// TIA Portal V18 export
// export: Created 2026-06-21T12:15:02Z, ExportSetting WithDefaults
PlcWatchTable "WT_PLC1_PID_VFD"
  PlcWatchTableEntry "HMI_Sim_Mode"
  PlcWatchTableEntry "PLC1_Loi_Tong"
  PlcWatchTableEntry "PLC1_EStop_Latch"
  PlcWatchTableEntry "PLC1_Loi_Dry_Run"
  PlcWatchTableEntry "PLC1_Loi_Dosing"
  PlcWatchTableEntry "PLC1_Loi_Truyen_Thong"
  PlcWatchTableEntry "PLC1_Loi_Setpoint"
  PlcWatchTableEntry "BonChua_Loi_Setpoint"
  PlcWatchTableEntry "PID_Bon2_Error"
  PlcWatchTableEntry "PID_Bon2_ErrorBits"
  PlcWatchTableEntry "VFD_Bon2_MB_Error"
  PlcWatchTableEntry "Gia_Lap_Mat_Ket_Noi_HMI"
